// TIA Portal V21 export
DATA_BLOCK "Pht_Block"   // DB1230
// stored: InstanceOfName PHT Block, InstanceOfType FB
"PHT Block"
   // VAR_INPUT
   //    Secs : Bool;
   //    Start : Bool;
   //    Stop : Bool;
   //    Abort : Bool;
   //    AlarmAck : Bool;
   //    AlwaysTrue : Bool;
   //    StartupMsgSelection : Bool;
   //    spare1 : Bool;
   //    spare2 : Bool;
   //    EndMsgSelection : Bool;
   //    EndMsgAck : Bool;
   //    Fault : Bool;
   //    Popup1Enable : Bool;
   //    Popup2Enable : Bool;
   //    ScadaHmi : Bool;
   //    StabilizeTime : Int;
   //    SetPressure : Real;
   //    ReleasePressure : Real;
   //    FailPressure : Real;
   //    AcceptableLeakage : Real;
   //    HoldTime : Int;
   //    UtilityValveDelay : Int;
   //    "Actual Minimum Pressure" : Real;
   //    "Actual Maximum Pressure" : Real;
   //    MaximumAttemptToFailedSelection : Int;
   //    MaximumNoAttemptToFailed : Int;
   //    PrintInterval : Int;
   // END_VAR
   // VAR_OUTPUT
   //    StartupMsg1 : Bool;
   //    CycleOver : Bool;
   //    LineValves : Bool;
   //    ControlValve : Bool;
   //    UtilityValve : Bool;
   //    StartupMsg : Bool;
   //    EndMsg : Bool;
   //    TestPassAlarm : Bool;
   //    TestFailAlarm : Bool;
   //    DrainValves : Bool;
   //    StartupMsg2 : Bool;
   //    StabilizeActualSecs : DInt;
   //    HoldActualMins : DInt;
   //    HoldActualSecs : DInt;
   //    Status : Int;
   //    StatusStr : String[60];
   //    UtilityValveActualDelay : Int;
   //    Event : Word;
   // END_VAR
   // VAR_IN_OUT
   //    Selected : Bool;
   //    CycleSelected : Bool;
   //    Running : Bool;
   //    VesselPressurised : Bool;
   //    DataLogCmd : Bool;
   //    StartLog : Bool;
   //    EndLog : Bool;
   //    DataLogYes : Bool;
   //    ResetPhtTimer : Bool;
   //    VesselStabilised : Bool;
   //    DelayToConfirmVesselPressurized : Bool;
   //    PressureDropDuringStabilizeTime : Bool;
   //    PressureDropDuringHoldTime : Bool;
   //    TestPassedRW : Bool;
   //    DelayToStartReleaseDone : Bool;
   //    DrainValve : Bool;
   //    StabilizePopup : Bool;
   //    LineValvesOpeningTime : Int;
   //    DrainValvesOpeningTime : Int;
   //    AcceptablePressure : Real;
   //    "PHT Selected" : Bool;
   //    TestAborted : Bool;
   //    ResetBit : Bool;
   //    Popup2Ack : Bool;
   //    StartupMsgYes : Bool;
   //    StartupMsgNo : Bool;
   //    MaximumNoAttemptToFailedTemp : Int;
   // END_VAR
   // VAR
   //    StabilizeTimer { S7_SetPoint := 'True'} : "R_TIMER";
   //    HoldTimer { S7_SetPoint := 'True'} : "R_TIMER";
   //    CheckPressureDuringStabilizeTime { S7_SetPoint := 'True'} : "On Delay Timer";
   //    CheckPressureDuringHoldTime { S7_SetPoint := 'True'} : "On Delay Timer";
   //    ReleaseCheckTime { S7_SetPoint := 'True'} : "On Delay Timer";
   //    CheckPressuredelay { S7_SetPoint := 'True'} : "On Delay Timer";
   //    DelayToStartRelease { S7_SetPoint := 'True'} : "On Delay Timer";
   //    StabilizeDelay { S7_SetPoint := 'True'} : "On Delay Timer";
   //    IEC_Timer_0_Instance { S7_SetPoint := 'True'} : TON_TIME;
   //    IEC_Timer_1_Instance { S7_SetPoint := 'True'} : TON_TIME;
   //    Timer1 { S7_SetPoint := 'True'} : TON_TIME;
   //    Timer2 { S7_SetPoint := 'True'} : TON_TIME;
   //    Timer3 { S7_SetPoint := 'True'} : TON_TIME;
   //    Timer4 { S7_SetPoint := 'True'} : TON_TIME;
   //    Timer5 { S7_SetPoint := 'True'} : TON_TIME;
   //    Timer6 { S7_SetPoint := 'True'} : TON_TIME;
   //    Timer7 { S7_SetPoint := 'True'} : TON_TIME;
   //    Re { ExternalAccessible := 'False'; ExternalVisible := 'False'; ExternalWritable := 'False'} : Bool;
   //    Re1 { ExternalAccessible := 'False'; ExternalVisible := 'False'; ExternalWritable := 'False'} : Bool;
   //    Re2 { ExternalAccessible := 'False'; ExternalVisible := 'False'; ExternalWritable := 'False'} : Bool;
   //    Re3 { ExternalAccessible := 'False'; ExternalVisible := 'False'; ExternalWritable := 'False'} : Bool;
   //    Re4 { ExternalAccessible := 'False'; ExternalVisible := 'False'; ExternalWritable := 'False'} : Bool;
   //    Re5 { ExternalAccessible := 'False'; ExternalVisible := 'False'; ExternalWritable := 'False'} : Bool;
   //    Re6 { ExternalAccessible := 'False'; ExternalVisible := 'False'; ExternalWritable := 'False'} : Bool;
   //    Re7 { ExternalAccessible := 'False'; ExternalVisible := 'False'; ExternalWritable := 'False'} : Bool;
   //    Re8 { ExternalAccessible := 'False'; ExternalVisible := 'False'; ExternalWritable := 'False'} : Bool;
   //    Re9 { ExternalAccessible := 'False'; ExternalVisible := 'False'; ExternalWritable := 'False'} : Bool;
   //    Re10 : Bool;
   //    Re11 : Bool;
   //    Re12 : Bool;
   //    Timer8 : TON_TIME;
   //    Timer9 { S7_SetPoint := 'True'} : TON_TIME;
   //    Timer10 { S7_SetPoint := 'True'} : TON_TIME;
   //    Timer11 { S7_SetPoint := 'True'} : TON_TIME;
   //    Timer12 { S7_SetPoint := 'True'} : TON_TIME;
   //    IEC_Counter_0_Instance { S7_SetPoint := 'True'} : CTU_INT;
   //    Re13 : Bool;
   //    Re14 : Bool;
   //    Re15 : Bool;
   //    timer13 : TON_TIME;
   // END_VAR
BEGIN
END_DATA_BLOCK
